// TIA Portal V17 export
// export: Created 2023-06-23T18:33:40.3624272Z, ExportSetting WithDefaults, DisplayName Totally Integrated Automation Portal, DisplayVersion V17, DisplayName TIA Portal Openness, DisplayVersion V17, DisplayName TIA Portal Version Control Interface, DisplayVersion V17, DisplayName STEP 7 Professional, DisplayVersion V17, DisplayName STEP 7 Safety, DisplayVersion V17, DisplayName WinCC Advanced / Unified PC, DisplayVersion V17
VAR_GLOBAL   // PLC tag table "22_AER-SP2"
   "iAER-SP2p" AT %I12.6 : Bool;   // 2
   "iAER-SP2" AT %I12.7 : Bool;   // 2
   "iAER-SP2a" AT %I20.1 : Bool;
   "oAER-SP2p" AT %Q12.1 : Bool;
   "oAER-SP2" AT %Q12.2 : Bool;
END_VAR
